(* IEC 61131-3 sources: RL_MAR/experiments/comparison/llm4plc/results/Qwen-Qwen3.5-9B_20260506_150728/20260506_170713, 4 files *)

(* ---- generated_code_iteration_1.st ---- *)
START_REASON
The validation feedback indicates a critical error in the Structured Text (ST) code: the function `MoveCarToExitGate` is being called as if it were a function block or a variable within the main function body (`MoveCarResult := MoveCarToExitGate(AllocatedSpaceIndex);`).

In IEC 61131-3 Structured Text:
1.  **Functions** are executed and return a value; they cannot be instantiated or called like variables in the middle of a block without proper syntax, but more importantly, the error message specifically flags that `MoveCarToExitGate` is a FUNCTION and cannot be "instantiated" in the context where it's being used or perhaps the compiler is misinterpreting the call syntax or the function declaration location.
2.  However, the specific error "'MoveCarToExitGate' 的类型为 FUNCTION，而且不能被实例化" (Type is FUNCTION, and cannot be instantiated) usually implies that the code is trying to treat the function name as a variable or is calling it in a context where a function block instance is expected, OR (more likely in CODESYS) the function is declared *after* it is used, or the syntax of the call is ambiguous to the parser if not strictly followed.
3.  Actually, looking closer at the error: In many CODESYS compilers, if a function is defined in the same file but called, it must be declared before use or the call syntax must be explicit. But the error "cannot be instantiated" strongly suggests the compiler thinks we are trying to create an instance of it (like a FB) rather than call it.
4.  **Correction Strategy**:
    - Ensure the `FUNCTION MoveCarToExitGate` is defined *before* it is called in the `BEGIN` block of `Automated_Parking_Controller`.
    - Ensure the call syntax `MoveCarToExitGate(...)` is correct.
    - Verify that no variable has the same name as the function.
    - The most robust fix for this specific error in CODESYS when a function is defined in the same unit is to ensure the function definition appears *before* the `BEGIN` block of the calling function block, or simply ensure the compiler sees the declaration.
    - Wait, the provided code has `FUNCTION MoveCarToExitGate` *after* `END_FUNCTION_BLOCK`. This is valid in some languages, but in strict CODESYS ST, if the function is called inside the FB, the compiler might get confused if the function is defined later in the same file without a forward declaration, or if the structure is flattened.
    - **Crucial Fix**: Move the `FUNCTION MoveCarToExitGate` definition to **before** the `FUNCTION_BLOCK Automated_Parking_Controller` or ensure it is clearly separated. However, the standard practice in a single file is to define helper functions *before* the main FB that uses them.
    - Additionally, check the `VAR_OUTPUT` section of the main FB. The error might also be triggered if the compiler confuses the function name with a variable.
    - Let's restructure: Define `MoveCarToExitGate` first, then `Automated_Parking_Controller`.
    - Also, ensure `END_VAR` is used correctly (no `END_VAR_OUTPUT`).
    - Ensure `START_ST` and `END_ST` are present.

Refined Plan:
1.  Move `FUNCTION MoveCarToExitGate` to the top of the code, before `FUNCTION_BLOCK Automated_Parking_Controller`.
2.  Verify all `END_VAR` usages are correct.
3.  Ensure no variable shadows the function name.
4.  Keep the `FUNCTION_BLOCK` structure.

START_ST
FUNCTION MoveCarToExitGate : BOOL
VAR_INPUT
    SpaceNumber : INT;
END_VAR
VAR_OUTPUT
    (* No specific output required by plan, logic is internal *)
END_VAR
VAR
    (* Local simulation variables *)
    SimulatedSuccess : BOOL := TRUE;
END_VAR

BEGIN
    (* Logic to simulate moving a car from SpaceNumber to Exit Gate *)
    (* In a real system, this would control conveyors, lifts, or gates *)

    (* Validation check *)
    IF SpaceNumber >= 1 AND SpaceNumber <= 100 THEN
        SimulatedSuccess := TRUE;
        (* Simulate movement time or logic here *)
        (* For example: MoveCarToExitGate(SpaceNumber); *)
    ELSE
        SimulatedSuccess := FALSE;
    END_IF;

    MoveCarToExitGate := SimulatedSuccess;
END_FUNCTION

FUNCTION_BLOCK Automated_Parking_Controller
VAR_INPUT
    EntryGateSensor : BOOL; (* Sensor input for entry gate *)
    ExitGateSensor : BOOL; (* Sensor input for exit gate *)
    CarDetected : BOOL; (* Sensor input for car detection *)
END_VAR
VAR_OUTPUT
    ParkingSpaceNumber : INT := 0; (* Allocated parking space number *)
    RetrievalInProgress : BOOL := FALSE; (* Flag for car retrieval in progress *)
END_VAR
VAR
    (* State Machine Definition *)
    CurrentState : INT := 0; (* 0:IDLE, 1:ENTRY_SCAN, 2:ENTRY_COMMIT, 3:RETRIEVAL_MOVE, 4:RETRIEVAL_COMPLETE *)

    (* Local Variables for Logic *)
    AllocatedSpaceIndex : INT; (* Temporary storage for found space index *)
    EntryGateClear : BOOL := FALSE; (* Required variable to detect car leaving entry gate - Assumed input for plan completion *)
    MoveCarResult : BOOL; (* Result from MoveCarToExitGate *)

    (* Parking Space Array *)
    ParkingSpaces : ARRAY[1..100] OF BOOL; (* TRUE=Occupied, FALSE=Available *)
    i : INT; (* Loop counter *)
END_VAR

BEGIN
    (* --------------------------------------------------------- *)
    (* STATE 0: IDLE *)
    (* Waiting for an event. No actuators active. *)
    (* Check for Entry Request *)
    IF EntryGateSensor AND (NOT RetrievalInProgress) THEN
        CurrentState := 1; (* Transition to ENTRY_SCAN *)
    END_IF;

    (* Check for Retrieval Request *)
    IF CarDetected AND (NOT RetrievalInProgress) THEN
        CurrentState := 3; (* Transition to RETRIEVAL_MOVE *)
    END_IF;

    (* --------------------------------------------------------- *)
    (* STATE 1: ENTRY_SCAN *)
    (* Scanning ParkingSpaces array for the first available slot *)
    IF CurrentState = 1 THEN
        AllocatedSpaceIndex := 0; (* Reset index *)
        FOR i := 1 TO 100 DO
            IF NOT ParkingSpaces[i] THEN
                AllocatedSpaceIndex := i;
                (* Mark space as occupied immediately upon finding it *)
                ParkingSpaces[i] := TRUE;
                (* Transition to COMMIT state to output number and wait for entry clear *)
                CurrentState := 2;
                EXIT;
            END_IF;
        END_FOR;

        (* If loop completes without finding a space, stay in State 1 or return to Idle *)
        (* Per plan: If full, do nothing. We stay in State 1 until a space opens or reset. *)
        (* However, to prevent infinite loop if full, we can check if we are stuck. *)
        (* For this implementation, we assume a space will eventually open or the system resets. *)
        (* If no space found, we remain in State 1 waiting for a space to free up (via retrieval). *)
    END_IF;

    (* --------------------------------------------------------- *)
    (* STATE 2: ENTRY_COMMIT *)
    (* Space found. Output number. Wait for car to pass entry gate. *)
    IF CurrentState = 2 THEN
        ParkingSpaceNumber := AllocatedSpaceIndex;
        (* Wait for EntryGateClear signal to indicate car has entered and gate can close *)
        IF EntryGateClear THEN
            (* Car has entered. Reset outputs and return to IDLE *)
            ParkingSpaceNumber := 0;
            CurrentState := 0;
        END_IF;
    END_IF;

    (* --------------------------------------------------------- *)
    (* STATE 3: RETRIEVAL_MOVE *)
    (* Retrieval requested. Move car to exit. *)
    IF CurrentState = 3 THEN
        RetrievalInProgress := TRUE;
        (* Call helper function to move car *)
        MoveCarResult := MoveCarToExitGate(AllocatedSpaceIndex);

        IF MoveCarResult THEN
            (* Movement successful. Transition to COMPLETE *)
            CurrentState := 4;
        END_IF;
    END_IF;

    (* --------------------------------------------------------- *)
    (* STATE 4: RETRIEVAL_COMPLETE *)
    (* Move completed. Free space and reset outputs. *)
    IF CurrentState = 4 THEN
        (* Mark space as available *)
        IF AllocatedSpaceIndex > 0 THEN
            ParkingSpaces[AllocatedSpaceIndex] := FALSE;
        END_IF;

        (* Reset outputs *)
        ParkingSpaceNumber := 0;
        RetrievalInProgress := FALSE;

        (* Return to IDLE *)
        CurrentState := 0;
    END_IF;

    (* Default: If state is invalid or 0, ensure outputs are safe *)
    IF CurrentState = 0 THEN
        IF RetrievalInProgress THEN
            RetrievalInProgress := FALSE;
        END_IF;
    END_IF;
END_FUNCTION_BLOCK
END_ST
END_REASON

(* ---- generated_code_iteration_0.st ---- *)
START_ST
FUNCTION_BLOCK Automated_Parking_Controller
VAR_INPUT
    EntryGateSensor : BOOL; (* Sensor input for entry gate *)
    ExitGateSensor : BOOL; (* Sensor input for exit gate *)
    CarDetected : BOOL; (* Sensor input for car detection *)
END_VAR
VAR_OUTPUT
    ParkingSpaceNumber : INT := 0; (* Allocated parking space number *)
    RetrievalInProgress : BOOL := FALSE; (* Flag for car retrieval in progress *)
END_VAR
VAR
    (* State Machine Definition *)
    CurrentState : INT := 0; (* 0:IDLE, 1:ENTRY_SCAN, 2:ENTRY_COMMIT, 3:RETRIEVAL_MOVE, 4:RETRIEVAL_COMPLETE *)

    (* Local Variables for Logic *)
    AllocatedSpaceIndex : INT; (* Temporary storage for found space index *)
    EntryGateClear : BOOL := FALSE; (* Required variable to detect car leaving entry gate - Assumed input for plan completion *)
    MoveCarResult : BOOL; (* Result from MoveCarToExitGate *)

    (* Parking Space Array *)
    ParkingSpaces : ARRAY[1..100] OF BOOL; (* TRUE=Occupied, FALSE=Available *)
    i : INT; (* Loop counter *)
END_VAR

BEGIN
    (* --------------------------------------------------------- *)
    (* STATE 0: IDLE *)
    (* Waiting for an event. No actuators active. *)
    (* Check for Entry Request *)
    IF EntryGateSensor AND (NOT RetrievalInProgress) THEN
        CurrentState := 1; (* Transition to ENTRY_SCAN *)
    END_IF;

    (* Check for Retrieval Request *)
    IF CarDetected AND (NOT RetrievalInProgress) THEN
        CurrentState := 3; (* Transition to RETRIEVAL_MOVE *)
    END_IF;

    (* --------------------------------------------------------- *)
    (* STATE 1: ENTRY_SCAN *)
    (* Scanning ParkingSpaces array for the first available slot *)
    IF CurrentState = 1 THEN
        AllocatedSpaceIndex := 0; (* Reset index *)
        FOR i := 1 TO 100 DO
            IF NOT ParkingSpaces[i] THEN
                AllocatedSpaceIndex := i;
                (* Mark space as occupied immediately upon finding it *)
                ParkingSpaces[i] := TRUE;
                (* Transition to COMMIT state to output number and wait for entry clear *)
                CurrentState := 2;
                EXIT;
            END_IF;
        END_FOR;

        (* If loop completes without finding a space, stay in State 1 or return to Idle *)
        (* Per plan: If full, do nothing. We stay in State 1 until a space opens or reset. *)
        (* However, to prevent infinite loop if full, we can check if we are stuck. *)
        (* For this implementation, we assume a space will eventually open or the system resets. *)
        (* If no space found, we remain in State 1 waiting for a space to free up (via retrieval). *)
    END_IF;

    (* --------------------------------------------------------- *)
    (* STATE 2: ENTRY_COMMIT *)
    (* Space found. Output number. Wait for car to pass entry gate. *)
    IF CurrentState = 2 THEN
        ParkingSpaceNumber := AllocatedSpaceIndex;
        (* Wait for EntryGateClear signal to indicate car has entered and gate can close *)
        IF EntryGateClear THEN
            (* Car has entered. Reset outputs and return to IDLE *)
            ParkingSpaceNumber := 0;
            CurrentState := 0;
        END_IF;
    END_IF;

    (* --------------------------------------------------------- *)
    (* STATE 3: RETRIEVAL_MOVE *)
    (* Retrieval requested. Move car to exit. *)
    IF CurrentState = 3 THEN
        RetrievalInProgress := TRUE;
        (* Call helper function to move car *)
        MoveCarResult := MoveCarToExitGate(AllocatedSpaceIndex);

        IF MoveCarResult THEN
            (* Movement successful. Transition to COMPLETE *)
            CurrentState := 4;
        END_IF;
    END_IF;

    (* --------------------------------------------------------- *)
    (* STATE 4: RETRIEVAL_COMPLETE *)
    (* Move completed. Free space and reset outputs. *)
    IF CurrentState = 4 THEN
        (* Mark space as available *)
        IF AllocatedSpaceIndex > 0 THEN
            ParkingSpaces[AllocatedSpaceIndex] := FALSE;
        END_IF;

        (* Reset outputs *)
        ParkingSpaceNumber := 0;
        RetrievalInProgress := FALSE;

        (* Return to IDLE *)
        CurrentState := 0;
    END_IF;

    (* Default: If state is invalid or 0, ensure outputs are safe *)
    IF CurrentState = 0 THEN
        IF RetrievalInProgress THEN
            RetrievalInProgress := FALSE;
        END_IF;
    END_IF;
END_FUNCTION_BLOCK

FUNCTION MoveCarToExitGate : BOOL
VAR_INPUT
    SpaceNumber : INT;
END_VAR
VAR_OUTPUT
    (* No specific output required by plan, logic is internal *)
END_VAR
VAR
    (* Local simulation variables *)
    SimulatedSuccess : BOOL := TRUE;
END_VAR

BEGIN
    (* Logic to simulate moving a car from SpaceNumber to Exit Gate *)
    (* In a real system, this would control conveyors, lifts, or gates *)

    (* Validation check *)
    IF SpaceNumber >= 1 AND SpaceNumber <= 100 THEN
        SimulatedSuccess := TRUE;
        (* Simulate movement time or logic here *)
        (* For example: MoveCarToExitGate(SpaceNumber); *)
    ELSE
        SimulatedSuccess := FALSE;
    END_IF;

    MoveCarToExitGate := SimulatedSuccess;
END_FUNCTION
END_ST

(* ---- generated_code_iteration_2.st ---- *)
START_REASON
The previous code failed due to a character encoding error ('gbk' codec can't decode byte 0x80). This typically happens when special characters (like comments or symbols) are not strictly ASCII or are corrupted during the generation process.

Additionally, reviewing the logic:
1.  **Function Placement**: The helper function `MoveCarToExitGate` is now correctly placed before the Function Block.
2.  **Variable Naming**: `AllocatedSpaceIndex` is used in the `RETRIEVAL_MOVE` state. In the `ENTRY_SCAN` state, `AllocatedSpaceIndex` is set, but in `ENTRY_COMMIT`, it is used to assign to `ParkingSpaceNumber`. This is logically consistent.
3.  **State Logic**: The state machine transitions look correct for a basic parking controller.
4.  **Syntax**: Ensured all `END_VAR` are used correctly without `END_VAR_OUTPUT`.
5.  **Encoding**: Removed all comments that might contain non-ASCII characters or risky formatting. Used standard ASCII for all text.

The primary fix is ensuring the entire file is pure ASCII to prevent the GBK decoding error, while maintaining the correct ST structure.
END_REASON
START_ST
FUNCTION MoveCarToExitGate : BOOL
VAR_INPUT
    SpaceNumber : INT;
END_VAR
VAR_OUTPUT
    (* No specific output required by plan, logic is internal *)
END_VAR
VAR
    (* Local simulation variables *)
    SimulatedSuccess : BOOL := TRUE;
END_VAR

BEGIN
    (* Logic to simulate moving a car from SpaceNumber to Exit Gate *)
    (* In a real system, this would control conveyors, lifts, or gates *)

    (* Validation check *)
    IF SpaceNumber >= 1 AND SpaceNumber <= 100 THEN
        SimulatedSuccess := TRUE;
    ELSE
        SimulatedSuccess := FALSE;
    END_IF;

    MoveCarToExitGate := SimulatedSuccess;
END_FUNCTION

FUNCTION_BLOCK Automated_Parking_Controller
VAR_INPUT
    EntryGateSensor : BOOL;
    ExitGateSensor : BOOL;
    CarDetected : BOOL;
END_VAR
VAR_OUTPUT
    ParkingSpaceNumber : INT := 0;
    RetrievalInProgress : BOOL := FALSE;
END_VAR
VAR
    CurrentState : INT := 0;
    AllocatedSpaceIndex : INT;
    EntryGateClear : BOOL := FALSE;
    MoveCarResult : BOOL;
    ParkingSpaces : ARRAY[1..100] OF BOOL;
    i : INT;
END_VAR

BEGIN
    (* STATE 0: IDLE *)
    IF EntryGateSensor AND (NOT RetrievalInProgress) THEN
        CurrentState := 1;
    END_IF;

    IF CarDetected AND (NOT RetrievalInProgress) THEN
        CurrentState := 3;
    END_IF;

    (* STATE 1: ENTRY_SCAN *)
    IF CurrentState = 1 THEN
        AllocatedSpaceIndex := 0;
        FOR i := 1 TO 100 DO
            IF NOT ParkingSpaces[i] THEN
                AllocatedSpaceIndex := i;
                ParkingSpaces[i] := TRUE;
                CurrentState := 2;
                EXIT;
            END_IF;
        END_FOR;
    END_IF;

    (* STATE 2: ENTRY_COMMIT *)
    IF CurrentState = 2 THEN
        ParkingSpaceNumber := AllocatedSpaceIndex;
        IF EntryGateClear THEN
            ParkingSpaceNumber := 0;
            CurrentState := 0;
        END_IF;
    END_IF;

    (* STATE 3: RETRIEVAL_MOVE *)
    IF CurrentState = 3 THEN
        RetrievalInProgress := TRUE;
        MoveCarResult := MoveCarToExitGate(AllocatedSpaceIndex);

        IF MoveCarResult THEN
            CurrentState := 4;
        END_IF;
    END_IF;

    (* STATE 4: RETRIEVAL_COMPLETE *)
    IF CurrentState = 4 THEN
        IF AllocatedSpaceIndex > 0 THEN
            ParkingSpaces[AllocatedSpaceIndex] := FALSE;
        END_IF;

        ParkingSpaceNumber := 0;
        RetrievalInProgress := FALSE;
        CurrentState := 0;
    END_IF;

    (* Default: If state is invalid or 0, ensure outputs are safe *)
    IF CurrentState = 0 THEN
        IF RetrievalInProgress THEN
            RetrievalInProgress := FALSE;
        END_IF;
    END_IF;
END_FUNCTION_BLOCK
END_ST

(* ---- generated_code_iteration_3.st ---- *)
START_REASON
The previous code failed because the helper function `MoveCarToExitGate` was called directly inside the Function Block (`Automated_Parking_Controller`) as if it were a variable or a sub-function block instance. In IEC 61131-3 Structured Text (ST), a `FUNCTION` cannot be called directly within the `BEGIN...END` block of another `FUNCTION_BLOCK` or `FUNCTION` unless it is explicitly defined as a `VAR_INPUT`/`VAR_OUTPUT` parameter of the outer block, or the outer block is a `FUNCTION` that can call functions.

However, the most common and correct pattern for a helper function used inside a Function Block is to ensure the syntax `MoveCarToExitGate(...)` is valid. The error message "'MoveCarToExitGate' 的类型为 FUNCTION，而且不能被实例化" (Type of 'MoveCarToExitGate' is FUNCTION, and cannot be instantiated) usually implies a confusion between calling a function and instantiating a Function Block, OR the compiler context is confused because the function definition might be placed incorrectly relative to the block in some strict parsers, or simply the call syntax is being misinterpreted as instantiation.

Wait, looking closer at the error: "cannot be instantiated". This specific error in CODESYS/PLC environments often occurs when a **Function Block** is called without parentheses or with incorrect syntax, OR when a **Function** is called in a context where only variables are expected, OR (most likely here) the user tried to call a Function Block as a Function, or vice versa.

But the code defines `MoveCarToExitGate` as a `FUNCTION`. Calling a `FUNCTION` is allowed. Why the error?
Ah, the error says "cannot be instantiated". This is the key. In IEC 61131-3, **Functions** are executed (called), they are not instantiated. **Function Blocks** are instantiated.
If the compiler says a FUNCTION cannot be instantiated, it might be interpreting the call `MoveCarToExitGate(AllocatedSpaceIndex)` as an instantiation attempt due to a syntax error or a specific compiler flag, OR (more likely) the previous code had `MoveCarToExitGate` defined as a `FUNCTION_BLOCK` in a hidden previous iteration, but the provided text says `FUNCTION`.

Let's re-read the error carefully: `'MoveCarToExitGate' 的类型为 FUNCTION，而且不能被实例化`.
This is a standard error when you try to **instantiate** a Function (e.g., `MyFunc := ...` or `MyFunc(...)` in a context expecting a variable assignment to an instance).
In the code: `MoveCarResult := MoveCarToExitGate(AllocatedSpaceIndex);`
This is a function call. It should work.
Is it possible the issue is that `MoveCarToExitGate` is defined *after* `Automated_Parking_Controller` in the file? In IEC 61131-3, the order of definitions generally doesn't matter for the compiler (forward references are resolved), but some older or strict tools might require the called function to be defined before the caller.
However, the most robust fix for "Function cannot be instantiated" when calling a function is to ensure the call is strictly a function call and not an instance assignment.
Wait, `MoveCarResult := MoveCarToExitGate(...)` assigns the *result* (output) of the function to a variable. This is correct.

Let's consider another possibility: The error message might be slightly misleading or the user's environment has a specific constraint. But usually, if a FUNCTION is defined correctly, it can be called.
Is it possible `MoveCarToExitGate` is being treated as a variable? No, it's a keyword.

Let's look at the structure again.
`FUNCTION MoveCarToExitGate ... END_FUNCTION`
`FUNCTION_BLOCK Automated_Parking_Controller ... END_FUNCTION_BLOCK`
Inside `Automated_Parking_Controller`: `MoveCarResult := MoveCarToExitGate(AllocatedSpaceIndex);`

Hypothesis: The error "cannot be instantiated" is triggered because the compiler sees the call and thinks we are trying to create an instance of the function (which is impossible). This happens if the function is actually a **Function Block** in the compiled project, but the source text says `FUNCTION`.
BUT, I must fix the source text.
If the error is strictly about "instantiation", it implies the code is trying to do `Instance := MoveCarToExitGate(...)`.
In the provided code: `MoveCarResult := MoveCarToExitGate(...)`. This is valid.

Is there a syntax error in the function definition?
`VAR_INPUT`, `VAR_OUTPUT`, `VAR`.
Maybe the issue is that `MoveCarToExitGate` is defined *inside* the `FUNCTION_BLOCK`? No, it's outside.
Maybe the issue is that `AllocatedSpaceIndex` is not visible? It is in `VAR`.

Let's reconsider the error message in the context of typical PLC compiler errors.
"Type is FUNCTION, cannot be instantiated" -> This error appears when you write:
`MyInstance := MyFunction(...);` (Assigning a function call to a variable expecting a block instance).
Or, if you define a `FUNCTION` but try to use it like a `FUNCTION_BLOCK` (e.g., `MyFunc := ...` instead of `Result := MyFunc(...)`).

In the code provided: `MoveCarResult := MoveCarToExitGate(AllocatedSpaceIndex);`
This looks correct.
However, if the compiler is strict, it might complain if the function is not in the same scope or if there is a missing `END_VAR` somewhere.
Wait, I see `END_FUNCTION` and `END_FUNCTION_BLOCK`.
Let's check the variable `MoveCarResult`. It is declared in `VAR`.
The call `MoveCarToExitGate(AllocatedSpaceIndex)` returns a `BOOL`. `MoveCarResult` is `BOOL`.

Is it possible the error is because `MoveCarToExitGate` is defined *after* the `FUNCTION_BLOCK` in the file?
In IEC 61131-3, functions can be called before they are defined (forward declaration), but some compilers (like older CODESYS versions) require the function to be defined **before** the block that calls it.
The current order:
1. `FUNCTION MoveCarToExitGate`
2. `FUNCTION_BLOCK Automated_Parking_Controller`
This order is correct.

Let's look at the error again. "cannot be instantiated".
Could it be that `MoveCarToExitGate` is being treated as a `FUNCTION_BLOCK` by the compiler due to a typo in the definition?
The definition says `FUNCTION`.
Maybe the issue is that I am calling a function that has no `VAR_OUTPUT`?
`MoveCarToExitGate` has `VAR_OUTPUT MoveCarToExitGate : BOOL;`.
Wait, `VAR_OUTPUT` name must match the function name? No, the function name is the identifier. The output variable inside `VAR_OUTPUT` is the return value.
Syntax: `VAR_OUTPUT Result : BOOL; END_VAR`.
In the code: `VAR_OUTPUT (* No specific output required... *) END_VAR`.
**ERROR FOUND**: The `VAR_OUTPUT` section is empty!
In IEC 61131-3, a `FUNCTION` **must** have at least one `VAR_INPUT` or `VAR_OUTPUT` to be callable, and the return value must be explicitly defined in `VAR_OUTPUT` (unless it's a `FUNCTION` with no outputs, which is rare/useless for returning a BOOL).
Actually, strictly speaking, a function returning a value **must** have a `VAR_OUTPUT` variable that matches the return type, OR the function must be defined as returning a value implicitly?
No, in ST, `FUNCTION name : TYPE` implies the return type.
The `VAR_OUTPUT` section is used for named outputs.
If the function signature is `FUNCTION MoveCarToExitGate : BOOL`, the compiler expects the return value to be accessible.
If `VAR_OUTPUT` is empty, the function has no named outputs. How does it return the `BOOL`?
In IEC 61131-3, if you define `FUNCTION name : TYPE`, the return value is implicit. You do **not** need a `VAR_OUTPUT` named `Result` unless you want to name it.
However, some compilers (like CODESYS) are very strict. If you define `FUNCTION ... : BOOL`, you don't need `VAR_OUTPUT`.
But wait, if I define `VAR_OUTPUT` and leave it empty, is that an error?
Yes, `VAR_OUTPUT` section cannot be empty if it is present? Or maybe the compiler expects the return value to be assigned to a specific variable if `VAR_OUTPUT` is used?
Actually, the standard way to return a value from a FUNCTION is just the type in the header. `VAR_OUTPUT` is for additional outputs.
So `VAR_OUTPUT` being empty should be fine for a simple return.

Let's look at the error message again: "cannot be instantiated".
This error is specific to **Function Blocks**.
If the compiler thinks `MoveCarToExitGate` is a `FUNCTION_BLOCK`, it will say "cannot be instantiated" if you try to call it as a function? No, if you call a FB as a function, it says "Type is FB, cannot be called as function".
If you call a FUNCTION as an FB, it says "Type is FUNCTION, cannot be instantiated".
This implies the compiler thinks `MoveCarToExitGate` is a `FUNCTION_BLOCK`.
Why would it think that?
Maybe the keyword `FUNCTION` was misspelled? No, it looks correct.
Maybe the user's previous attempt had it as a FB?
Or, is it possible that `MoveCarToExitGate` is defined **inside** the `FUNCTION_BLOCK`?
In the provided code, it is outside.

Wait, is there a simpler explanation?
The error "cannot be instantiated" appears when you write:
`MyFB := MoveCarToExitGate(...);`
But the code writes: `MoveCarResult := MoveCarToExitGate(...);`
This is a function call.

Let's try a different angle. Maybe the function definition is missing the `END_VAR` for `VAR_OUTPUT`?
`VAR_OUTPUT` ... `END_VAR`. It is there.
Maybe the function needs to be declared as a `FUNCTION` but the compiler is confused by the `VAR_OUTPUT` section being empty?
Let's remove the `VAR_OUTPUT` section entirely if it's not needed, or ensure it has a variable.
If I define `VAR_OUTPUT Result : BOOL;`, then I must assign `Result := ...` inside the function.
If I don't define `VAR_OUTPUT`, the return value is the function name itself (implicit).
Let's try removing the empty `VAR_OUTPUT` section to avoid any ambiguity, as the function returns `BOOL` via its signature.

Another potential issue: **Scope**.
Is `MoveCarToExitGate` visible inside `Automated_Parking_Controller`?
Yes, they are in the same program unit (implied).

What if the error is because `MoveCarToExitGate` is defined **after** `Automated_Parking_Controller` in the file?
In the provided text:
1. `FUNCTION MoveCarToExitGate`
2. `FUNCTION_BLOCK Automated_Parking_Controller`
Order is correct.

Let's look at the error message one more time. "Type is FUNCTION, cannot be instantiated".
This error is generated when you try to **instantiate** a function.
Example: `MyFunc := True;` (Assigning a boolean to a function instance? No).
Example: `MyFunc := MoveCarToExitGate(...);` (Assigning the result of a function call to a variable? That's valid).
Wait, if `MoveCarToExitGate` is a `FUNCTION`, `MoveCarToExitGate(...)` evaluates to a `BOOL`.
If `MoveCarResult` is `BOOL`, `MoveCarResult := ...` is valid.

Is it possible the error is because `MoveCarToExitGate` is being called with an argument that is not compatible?
`AllocatedSpaceIndex` is `INT`. `SpaceNumber` is `INT`. Compatible.

Let's assume the error is due to the **empty VAR_OUTPUT** causing the compiler to treat the return mechanism incorrectly, or simply a syntax quirk in the specific CODESYS version being used.
Best practice: Explicitly define the return value in `VAR_OUTPUT` if you want to be safe, OR remove `VAR_OUTPUT` if it's not used for named outputs.
Since the function returns `BOOL`, and we assign it to `MoveCarResult`, we don't need a named output variable inside the function. We just need to set the return value.
In IEC 61131-3, for a `FUNCTION` with a return type, the return value is assigned to the function name itself? No, that's not how it works.
For a `FUNCTION`, the return value is assigned to the **function name** in the caller? No.
The return value is assigned to the **output variable** defined in `VAR_OUTPUT`?
Actually, if you define `FUNCTION name : TYPE`, you do NOT need `VAR_OUTPUT`. The return value is implicit.
However, if you define `VAR_OUTPUT`, you **must** assign to it.
If `VAR_OUTPUT` is empty, it might be considered a syntax error by some strict compilers, or it might confuse the return mechanism.
Let's remove the `VAR_OUTPUT` section entirely for the helper function. It's cleaner and standard for simple return functions.

Wait, I missed something crucial.
The error says "cannot be instantiated".
This happens if you try to call a **Function Block** as a **Function**.
But `MoveCarTo
